FUNCTION_BLOCK TRollingAverage
VAR_INPUT
END_VAR
VAR_OUTPUT
END_VAR
VAR
    pSamples : POINTER TO LREAL;
    SampleCount : UDINT;
    MaxSamples : UDINT;
END_VAR

METHOD AddSample
VAR_INPUT
    Value : LREAL;
END_VAR
IF pSamples > 0 THEN
    IF SampleCount < MaxSamples THEN
        pSamples[SampleCount] := Value;
        SampleCount := SampleCount + 1;
    ELSE
        MEMMOVE(
            destAddr := ADR(pSamples[0]),
            srcAddr  := ADR(pSamples[1]),
            n        := SIZEOF(pSamples[0]) * (MaxSamples-1));
        pSamples[MaxSamples - 1] := Value;
    END_IF
END_IF
END_METHOD

METHOD Clear
VAR_INPUT
END_VAR
IF pSamples > 0 THEN
    MEMSET(
        destAddr := pSamples,
        fillByte := 0,
        n        := MaxSamples * SIZEOF(pSamples[0]));
        
    SampleCount := 0;
END_IF
END_METHOD

METHOD FB_exit : BOOL
VAR_INPUT
	bInCopyCode : BOOL; // if TRUE, the exit method is called for exiting an instance that is copied afterwards (online change).
END_VAR
IF bInCopyCode = FALSE THEN // avoid deleting samples on online change!
    __DELETE(pSamples);
END_IF
END_METHOD

METHOD FB_init : BOOL
VAR_INPUT
	bInitRetains : BOOL; // if TRUE, the retain variables are initialized (warm start / cold start)
	bInCopyCode : BOOL;  // if TRUE, the instance afterwards gets moved into the copy code (online change)
    MaxSamples : UDINT;
END_VAR
pSamples := __NEW(LREAL,MaxSamples);
THIS^.MaxSamples := MaxSamples;
END_METHOD

METHOD GetAverage : LREAL
VAR
    i : UDINT;
    Sum : LREAL;
END_VAR
IF pSamples > 0 AND SampleCount > 0 THEN
    FOR i := 0 TO SampleCount - 1 DO
        Sum := Sum + pSamples[i];
    END_FOR
    GetAverage := Sum/SampleCount;
END_IF
END_METHOD

END_FUNCTION_BLOCK

(* stored: Version 1.1.0.1, ProductVersion 3.1.4024.3
   POU TRollingAverage: Id {accb748c-a23e-031b-313f-6e7939502a8e}, SpecialFunc None
   Method AddSample: Id {e0e47fcd-c523-0260-35a2-73a764a09a40}
   Method Clear: Id {c2ee7530-b6ad-0558-0d66-8cb678e191dc}
   Method FB_exit: Id {e933eafc-4652-0b34-34e7-ed6815d6d2e0}
   Method FB_init: Id {304218cd-9cf9-0959-0655-fd4d5e2df93e}
   Method GetAverage: Id {b54ae141-3192-06ad-07c8-620dac680633} *)
